FUNCTION fMembershipDegreeArray : REAL;
VAR
	i,j:DINT;
END_VAR
VAR_IN_OUT
	FisVariables:ARRAY[*]OF FIS_VAR;
	MD : ARRAY[*  , *  ] OF REAL;
//MD:ARRAY[*]OF ARRAY[*] OF REAL;
END_VAR
VAR_OUTPUT
	error: BOOL;
END_VAR

FOR i:=LOWER_BOUND(FisVariables,1) TO UPPER_BOUND(FisVariables,1) DO
	FOR j:=1 TO FisVariables[I].NumberOfMF DO
		MD[i,j]:= 
			fMembershipDegree(
				CrispInput := FisVariables[i].CrispValue,
				MD[i,j] := FisVariables[i].MF[j]);
	END_FOR	
END_FOR

END_FUNCTION

(* stored: Version 1.1.0.1, ProductVersion 3.1.4024.6
   POU fMembershipDegreeArray: Id {6d363a7a-af14-41e4-a352-af3263690f62}, SpecialFunc None *)
